// Mitsubishi GX Works2 project: 230927-009-exercicio final   PLC: Q03UDV

// task Task_01 (event TRUE, interval 0, priority 31): POU_01

PROGRAM POU_01
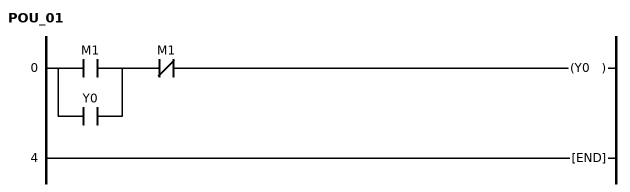
0     LD      M1
      OR      Y0
      ANI     M1
      OUT     Y0
4     END
END_PROGRAM
